// TIA Portal V16 export
// export: Created 2023-03-29T11:03:44.0749108Z, ExportSetting WithDefaults, DisplayName Totally Integrated Automation Portal, DisplayVersion V16 Update 6, DisplayName TIA Portal Version Control Interface, DisplayVersion V16 Update 2, DisplayName TIA Portal Openness, DisplayVersion V16 Update 6, DisplayName STEP 7 Professional, DisplayVersion V16 Update 6, DisplayName STEP 7 Safety, DisplayVersion V16, DisplayName WinCC Advanced, DisplayVersion V16 Update 6
VAR_GLOBAL   // PLC tag table "Tag HMI"
   "HMI.ManualMode_visible" AT %M1023.1 : Bool;
   "HMI.ErrorBits_Int" AT %MW1024 : Int;
   "HMI.Warning_Int" AT %MW1028 : Int;
   "HMI.ErrorAck_Int" AT %MW1026 : Int;
   ProcessMemory_Static_1_setChanging AT %M9.2 : Bool;   // Znacznik pobierania konfiguracji do instancji pamięci peocesu
   "HMI.Acknowledge_visible" AT %M1030.1 : Bool;
   memRis_WatchDog_HMI_PLC AT %M9.0 : Bool;
   "HMI.ErrorAck" AT %M1030.0 : Bool;
   "HMI.Filing3" AT %M1031.4 : Bool;   // bit informujący o wejściu w tryb napełniania
   "HMI.Warning_Int_tank" AT %MW1031 : Int;
   "HMI.rez" AT %M1031.1 : Bool;
   "HMI.StopFiling" AT %M1031.0 : Bool;   // bit informacji o zatrzymanym napełnianiu z powodu niskiego ciśnienia wna magistrali
   "HMI.Filing2" AT %M1031.3 : Bool;   // bit informujący o wejściu w tryb napełniania
   "HMI.Filing4" AT %M1031.5 : Bool;   // bit informujący o wejściu w tryb napełniania
   "HMI.Filing1" AT %M1031.2 : Bool;   // bit informujący o wejściu w tryb napełniania
END_VAR
